Universal Robots PolyScope program: MT_SPP_Template.urp

Program MT_SPP_Template (createdIn=3.5.1.10661 lastSavedIn=5.1.0.40195 robotSerialNumber=2014359999 directory=/home/ur/ursim-current/programs/Machine Tending/Card_Templates/SFF installation=default)
Calibrated DH parameters: a=[0, -0.425, -0.3922, 0, 0, 0]; d=[0.1625, 0, 0, 0.1333, 0.0997, 0.0996]; alpha=[1.570796, 0, 0, 1.570796, -1.570796, 0]; deltaTheta=[0, 0, 0, 0, 0, 0]
BeforeStart
  MoveJ speed 60 deg/s, acceleration 80 deg/s^2 (useActiveTCP=false) feature=Base
    Waypoint Wait_Machine: 
  Folder Status
    Infeed_Ready := True   [initializeExpression=False]
    Outfeed_Ready := True   [initializeExpression=False]
  Folder Initialization
    Call Tool_1_Off
Robot Program (runOnlyOnce=false)
  Wait Condition expression=Infeed_Ready≟ True
  Folder INFEED 
    MoveL speed 1000 mm/s, acceleration 2500 mm/s^2 (useActiveTCP=false) tcp=TCP; feature=Base
      Waypoint Pick_Approach: 
      Waypoint Pick_Position: 
      Call Tool_1_On
      Waypoint Pick_Approach: 
      Waypoint Wait_Machine: 
  Folder MACHINE
    'Wait for machine's "Request Load" '
    Wait Undefined
    Folder LOAD
      MoveL speed 1000 mm/s, acceleration 2500 mm/s^2 (useActiveTCP=false) tcp=TCP; feature=Base
        Waypoint Load_Approach: motionParameters(blendRadius=0.05)
        Waypoint Load_Position: 
        Call Holding_On
        Call Tool_1_Off
        Waypoint Load_Approach: 
        Waypoint Wait_Machine: 
      'Set "Load Complete" signal to High'
      Set Undefined
      'Wait "Request Load" reset (or some time) '
      Wait Undefined
      'Set "Load Complete" signal to Low'
      Set Undefined
    'Wait for machine's "Request Unload" '
    Wait Undefined
    Folder UNLOAD
      MoveL speed 1000 mm/s, acceleration 2500 mm/s^2 (useActiveTCP=false) tcp=TCP; feature=Base
        Waypoint Load_Approach: motionParameters(blendRadius=0.05)
        Waypoint Load_Position: 
        Call Tool_1_On
        Call Holding_Off
        Waypoint Load_Approach: 
        Waypoint Wait_Machine: 
      'Set "Unload Complete" signal to High'
      Set Undefined
      'Wait "Request Unload" reset (or some time) '
      Wait Undefined
      'Set "Unload Complete" signal to Low'
      Set Undefined
  Wait Condition expression=Outfeed_Ready≟ True
  Folder OUTFEED 
    MoveJ speed 120 deg/s, acceleration 150 deg/s^2 (useActiveTCP=false) tcp=TCP; feature=Base
      Waypoint Mach_to_Outfeed: motionParameters(blendRadius=0.05)
    MoveL speed 250 mm/s, acceleration 1200 mm/s^2 (useActiveTCP=false) tcp=TCP; feature=Base
      Waypoint Place_Approach: 
      Waypoint Place_Position: 
      Call Tool_1_Off
      Waypoint Place_Approach: 
SubProgram  [hidden by the author, left out]
SubProgram  [hidden by the author, left out]
SubProgram  [hidden by the author, left out]
SubProgram  [hidden by the author, left out]
SubProgram Tool_1_Off [hidden by the author, left out]
SubProgram Tool_1_On [hidden by the author, left out]
SubProgram Holding_On [hidden by the author, left out]
SubProgram Holding_Off [hidden by the author, left out]
